FUNCTION_BLOCK EL2574PixelReader IMPLEMENTS I_PixelReader
VAR
	pixelValue : TcVnVector4_LREAL;
END_VAR

METHOD PUBLIC ReadAsUdint : UDINT
VAR_INPUT
END_VAR

VAR
	pixel		: ARRAY[0..3] OF BYTE;
	pixelAsUint : UDINT;
END_VAR
pixel[0] := LREAL_TO_BYTE(value[0]);
pixel[1] := LREAL_TO_BYTE(value[1]);
pixel[2] := LREAL_TO_BYTE(value[2]);
//pixel[3] := LREAL_TO_BYTE(value[3]);
pixel[3]:=0;

memcpy(ADR(pixelAsUint), ADR(pixel),SIZEOF(pixelAsUint));
ReadAsUdint := pixelAsUint;
END_METHOD

PROPERTY PUBLIC Value : Reference to TcVnVector4_LREAL
GET
Value ref= pixelValue;
END_GET
END_PROPERTY

END_FUNCTION_BLOCK

(* stored: Version 1.1.0.1
   POU EL2574PixelReader: Id {e3e9ebcd-6c2d-4826-b14a-469ee1548339}, SpecialFunc None
   Method ReadAsUdint: Id {117163d6-f128-4391-95bb-ce0472d06b94}
   Property Value: Id {573b5eba-09d0-4305-827f-ce51c479cc62}
   Get Get: Id {7fd754e2-7be9-4e97-a852-5bd0386c6292} *)
